(* Logix 5000 project; controller PLCNo1 vendor 1 type 14 code 196 rev 35.11; software revision 35.00 *)

TASK MainTask (continuous, watchdog 500 ms) : MainProgram

MODULES
   Local : vendor 1 type 14 code 196 (5069 0, rev 35.11)
      PLCNo2 : vendor 1 type 14 code 196 (Ethernet 192.168.1.2, rev 35.1)
      ETAP : 1783-ETAP (Ethernet 192.168.1.101, rev 2.1)
      RPLC : 5094-AENTR (Ethernet 192.168.1.11, rev 4.1)
END_MODULES

PROGRAM MainProgram   (* main routine MainRoutine *)
VAR
   car_enter : BOOL;
   car_exit : BOOL;
   dry : BOOL;
   ons : SINT;
   post_rinse : BOOL;
   pre_rinse : BOOL;
   soap : BOOL;
   start : BOOL;
   stop : BOOL;
   Time : TIMER := (PRE := 61000);
   track_running : BOOL;
   washing : BOOL;
   wax : BOOL;
END_VAR

ROUTINE MainRoutine   (* ladder *)
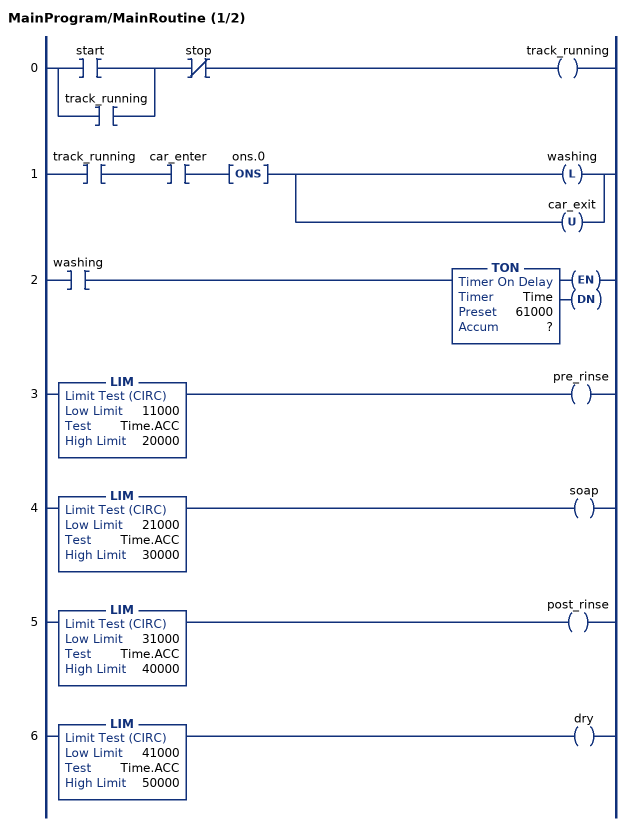
   0: [XIC(start) ,XIC(track_running) ]XIO(stop)OTE(track_running);
   1: XIC(track_running)XIC(car_enter)ONS(ons.0)[OTL(washing) ,OTU(car_exit) ];
   2: XIC(washing)TON(Time,?,?);
   3: LIM(11000,Time.ACC,20000)OTE(pre_rinse);
   4: LIM(21000,Time.ACC,30000)OTE(soap);
   5: LIM(31000,Time.ACC,40000)OTE(post_rinse);
   6: LIM(41000,Time.ACC,50000)OTE(dry);
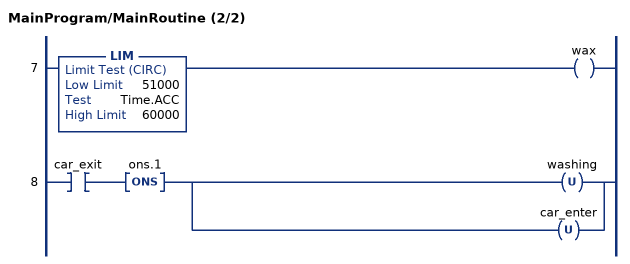
   7: LIM(51000,Time.ACC,60000)OTE(wax);
   8: XIC(car_exit)ONS(ons.1)[OTU(washing) ,OTU(car_enter) ];
END_ROUTINE
END_PROGRAM
